TYPE E_MessengerState :
(
	Init := 0,
	CreateSocket	:= 1,
	Active	:= 2,
	CloseSocket := 3,
	Error	:= 10
);
END_TYPE

(* stored: Version 1.1.0.1, ProductVersion 3.1.4018.5
   DUT E_MessengerState: Id {4bcf537e-a699-4180-bcfd-f772ea4b2b9e} *)
